{attribute 'qualified_only'}
{attribute 'strict'}
{attribute 'to_string'}
TYPE E_BridgeLinkStatus :
(
    Connected,                    // local State = OP, far device present, far side TxPDOState = 0 (OP)
    LocalNotOperational,          // local State <> OP
    RemoteNotConnected,   // far device not present
    RemoteNotOperational          // far device present but TxPDOState <> 0
) UDINT;
END_TYPE

(* stored: Version 1.1.0.1, ProductVersion 3.1.4024.12
   DUT E_BridgeLinkStatus: Id {0b2a777c-5a9d-4624-86df-f7f2aa9e3cab} *)
